Staubli VAL3: OnEvent11.pgx

program OnEvent11()
begin
  //-----------------------------------------------------------------------
  //Header begin
  //LasMAN3.7
  //Description of program
  //
  //Input parameters
  //
  //Output paramaters
  //Example
  //  call OnEvent1()
  //History
  //  Creation : 2013-06-23  y.ye@staubli.com
  //Header end
  //-----------------------------------------------------------------------
  //示教偏差
  resetMotion()
  call Teach:TeachOffset(DataBase:fOffset)
  DataBase:nInterfaceType=9
end
